// LS Electric XG5000 project: Tip-off System_230829-1
// 기종:PLC_K80S 제목: 회사: 저자: 설명: 
// PLC LSPLC
// module base 0 slot 0: 입출력 모듈:XBM-DN/DP32H2 (DC 24V입력/TR 출력, 32점)
// module base 0 slot 1: 내장위치결정:XBF-PO02E (오픈컬렉터형, 2축)
// module base 0 slot 2: 입력 모듈:XBE-DC16A/B (DC24V 입력, 16점 / DC12/24V 입력, 16점)
// module base 0 slot 3: 입력 모듈:XBE-DC16A/B (DC24V 입력, 16점 / DC12/24V 입력, 16점)
// module base 0 slot 4: 출력 모듈:XBE-RY16A (릴레이 출력, 16점 (2A용, 8점/COM))
// module base 0 slot 5: 출력 모듈:XBE-RY16A (릴레이 출력, 16점 (2A용, 8점/COM))

PROGRAM NewProgram (task: 스캔 프로그램)

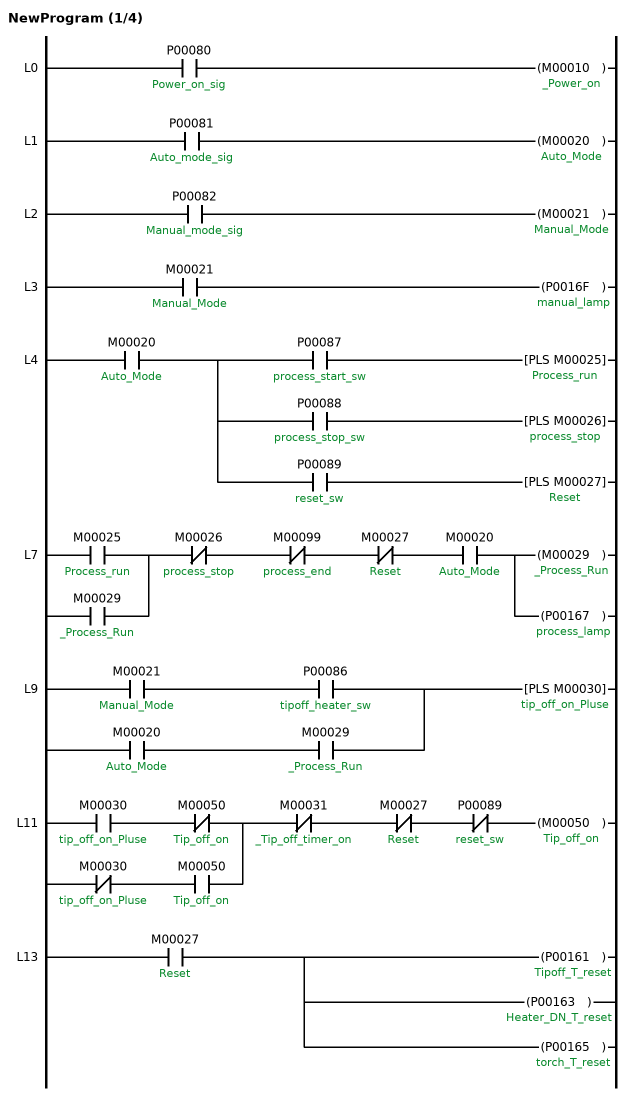
; L0
LOAD      P00080	// Power_on_sig
OUT       M00010	// _Power_on
; L1
LOAD      P00081	// Auto_mode_sig
OUT       M00020	// Auto_Mode
; L2
LOAD      P00082	// Manual_mode_sig
OUT       M00021	// Manual_Mode
; L3
LOAD      M00021	// Manual_Mode
OUT       P0016F	// manual_lamp
; L4
LOAD      M00020	// Auto_Mode
MPUSH
AND       P00087	// process_start_sw
OUTP      M00025	// Process_run
MLOAD
AND       P00088	// process_stop_sw
OUTP      M00026	// process_stop
MPOP
AND       P00089	// reset_sw
OUTP      M00027	// Reset
; L7
LOAD      M00025	// Process_run
OR        M00029	// _Process_Run
AND NOT   M00026	// process_stop
AND NOT   M00099	// process_end
AND NOT   M00027	// Reset
AND       M00020	// Auto_Mode
OUT       M00029	// _Process_Run
OUT       P00167	// process_lamp
; L9
LOAD      M00021	// Manual_Mode
AND       P00086	// tipoff_heater_sw
LOAD      M00020	// Auto_Mode
AND       M00029	// _Process_Run
OR LOAD
OUTP      M00030	// tip_off_on_Pluse
; L11
LOAD      M00030	// tip_off_on_Pluse
AND NOT   M00050	// Tip_off_on
LOAD NOT  M00030	// tip_off_on_Pluse
AND       M00050	// Tip_off_on
OR LOAD
AND NOT   M00031	// _Tip_off_timer_on
AND NOT   M00027	// Reset
AND NOT   P00089	// reset_sw
OUT       M00050	// Tip_off_on
; L13
LOAD      M00027	// Reset
OUT       P00161	// Tipoff_T_reset
OUT       P00163	// Heater_DN_T_reset
OUT       P00165	// torch_T_reset

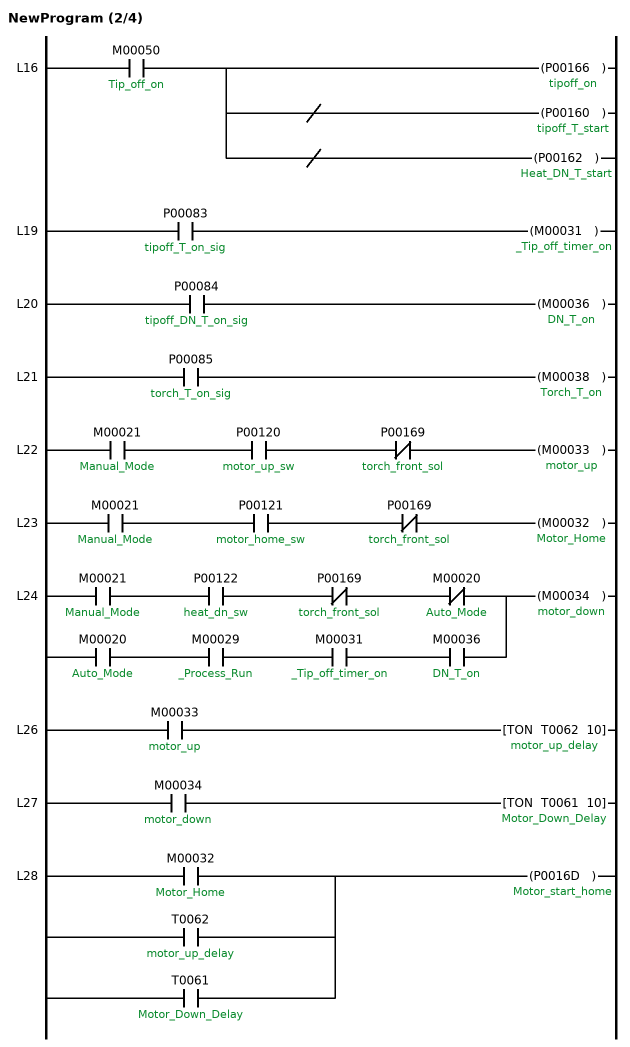
; L16
LOAD      M00050	// Tip_off_on
OUT       P00166	// tipoff_on
MPUSH
NOT
OUT       P00160	// tipoff_T_start
MPOP
NOT
OUT       P00162	// Heat_DN_T_start
; L19
LOAD      P00083	// tipoff_T_on_sig
OUT       M00031	// _Tip_off_timer_on
; L20
LOAD      P00084	// tipoff_DN_T_on_sig
OUT       M00036	// DN_T_on
; L21
LOAD      P00085	// torch_T_on_sig
OUT       M00038	// Torch_T_on
; L22
LOAD      M00021	// Manual_Mode
AND       P00120	// motor_up_sw
AND NOT   P00169	// torch_front_sol
OUT       M00033	// motor_up
; L23
LOAD      M00021	// Manual_Mode
AND       P00121	// motor_home_sw
AND NOT   P00169	// torch_front_sol
OUT       M00032	// Motor_Home
; L24
LOAD      M00021	// Manual_Mode
AND       P00122	// heat_dn_sw
AND NOT   P00169	// torch_front_sol
AND NOT   M00020	// Auto_Mode
LOAD      M00020	// Auto_Mode
AND       M00029	// _Process_Run
AND       M00031	// _Tip_off_timer_on
AND       M00036	// DN_T_on
OR LOAD
OUT       M00034	// motor_down
; L26
LOAD      M00033	// motor_up
TON       T0062 10	// motor_up_delay
; L27
LOAD      M00034	// motor_down
TON       T0061 10	// Motor_Down_Delay
; L28
LOAD      M00032	// Motor_Home
OR        T0062	// motor_up_delay
OR        T0061	// Motor_Down_Delay
OUT       P0016D	// Motor_start_home

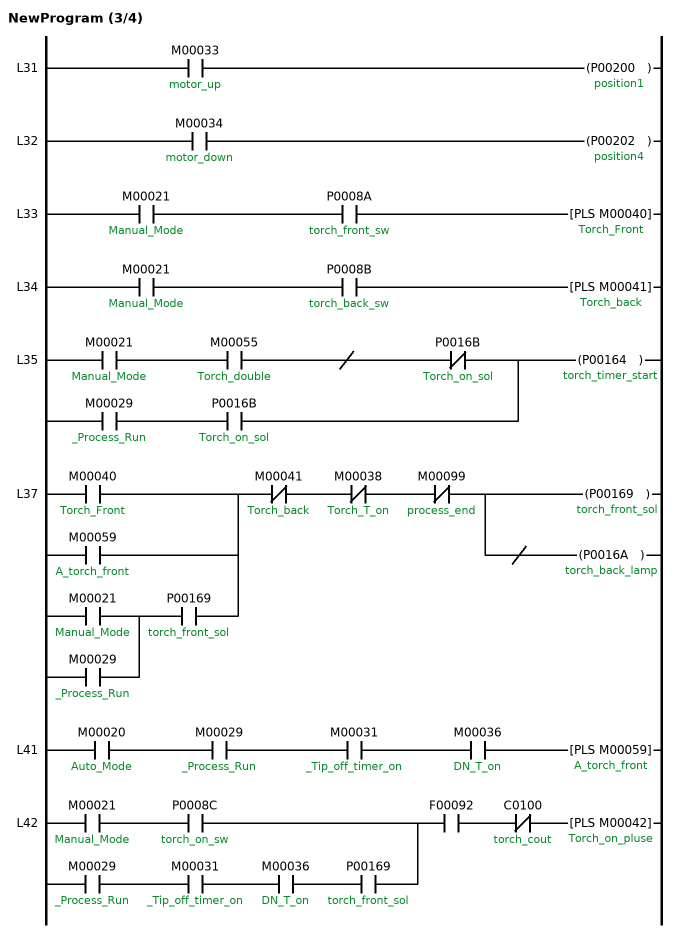
; L31
LOAD      M00033	// motor_up
OUT       P00200	// position1
; L32
LOAD      M00034	// motor_down
OUT       P00202	// position4
; L33
LOAD      M00021	// Manual_Mode
AND       P0008A	// torch_front_sw
OUTP      M00040	// Torch_Front
; L34
LOAD      M00021	// Manual_Mode
AND       P0008B	// torch_back_sw
OUTP      M00041	// Torch_back
; L35
LOAD      M00021	// Manual_Mode
AND       M00055	// Torch_double
NOT
AND NOT   P0016B	// Torch_on_sol
LOAD      M00029	// _Process_Run
AND       P0016B	// Torch_on_sol
OR LOAD
OUT       P00164	// torch_timer_start
; L37
LOAD      M00040	// Torch_Front
OR        M00059	// A_torch_front
LOAD      M00021	// Manual_Mode
OR        M00029	// _Process_Run
AND       P00169	// torch_front_sol
OR LOAD
AND NOT   M00041	// Torch_back
AND NOT   M00038	// Torch_T_on
AND NOT   M00099	// process_end
OUT       P00169	// torch_front_sol
NOT
OUT       P0016A	// torch_back_lamp
; L41
LOAD      M00020	// Auto_Mode
AND       M00029	// _Process_Run
AND       M00031	// _Tip_off_timer_on
AND       M00036	// DN_T_on
OUTP      M00059	// A_torch_front
; L42
LOAD      M00021	// Manual_Mode
AND       P0008C	// torch_on_sw
LOAD      M00029	// _Process_Run
AND       M00031	// _Tip_off_timer_on
AND       M00036	// DN_T_on
AND       P00169	// torch_front_sol
OR LOAD
AND       F00092
AND NOT   C0100	// torch_cout
OUTP      M00042	// Torch_on_pluse

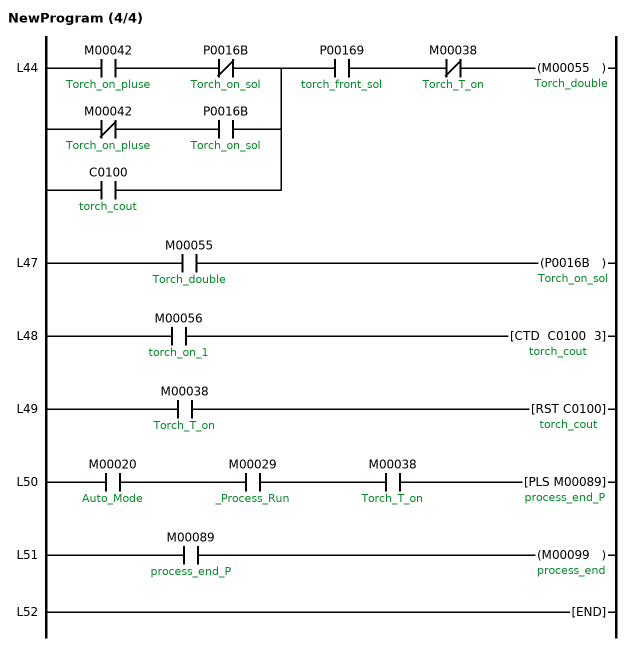
; L44
LOAD      M00042	// Torch_on_pluse
AND NOT   P0016B	// Torch_on_sol
LOAD NOT  M00042	// Torch_on_pluse
AND       P0016B	// Torch_on_sol
OR LOAD
OR        C0100	// torch_cout
AND       P00169	// torch_front_sol
AND NOT   M00038	// Torch_T_on
OUT       M00055	// Torch_double
; L47
LOAD      M00055	// Torch_double
OUT       P0016B	// Torch_on_sol
; L48
LOAD      M00056	// torch_on_1
CTD       C0100 3	// torch_cout
; L49
LOAD      M00038	// Torch_T_on
RST       C0100	// torch_cout
; L50
LOAD      M00020	// Auto_Mode
AND       M00029	// _Process_Run
AND       M00038	// Torch_T_on
OUTP      M00089	// process_end_P
; L51
LOAD      M00089	// process_end_P
OUT       M00099	// process_end
; L52
END

VARIABLES AND COMMENTS (devices not used above)
M00101	BIT	H_L_end
P00100	BIT	H_L_완료
M00105	BIT	H_R_end
T0101	BIT/WORD	H_R_start
M00103	BIT	L_H_end
T0100	BIT/WORD	L_H_start
M00067	BIT	Motor_DN_END
T0060	BIT/WORD	motor_homing_delay
P00055	BIT	motor_out_3
M00063	BIT	Motor_Run_DN_
M00064	BIT	Motor_run_up_
S00201	BIT	motor_step1_up_
S00202	BIT	motor_step2_dn_
S00203	BIT	motor_step3_up_
S00204	BIT	motor_step4_dn_
M00076	BIT	Motor_Strat
P00201	BIT	position2
M00028	BIT	Process_hold
T0081	BIT/WORD	step1_end
T0080	BIT/WORD	step1_start
T0083	BIT/WORD	step2_end
T0082	BIT/WORD	step2_start
T0085	BIT/WORD	step3_end
T0084	BIT/WORD	step3_start
T0087	BIT/WORD	step4_end
T0086	BIT/WORD	step4_start
M00080	BIT	step_start
T0070	BIT/WORD	tilie_H_L_end
M00071	BIT	tilite_Home
M00100	BIT	Tilite_H_L
M00070	BIT	tilite_L
M00102	BIT	Tilite_L_H
P0004D	BIT	Tilit_Home_sol
S00105	BIT	tilte_1_cycle
C0010	BIT/WORD	tilte_2_cycle
M00073	BIT	tilte_count
T0075	BIT/WORD	Tilte_end
P0000E	BIT	tilte_home_sw
S00101	BIT	Tilte_H_L
M00104	BIT	Tilte_H_R
T0072	BIT/WORD	tilte_H_R_end
P0000D	BIT	tilte_Left_sw
S00102	BIT	Tilte_L_H
T0071	BIT/WORD	Tilte_L_H_end
P0004C	BIT	Tilte_L_sol
S00100	BIT	Tilte_reset
M00072	BIT	tilte_right
P0004E	BIT	tilte_right_sol
P0000F	BIT	tilte_right_sw
S00104	BIT	Tilte_R_H
T0073	BIT/WORD	Tilte_R_H_end
M00085	BIT	torch_start
M00035	BIT	Up_Dn_Timer_on
M00062	BIT	_Motor_down
M00060	BIT	_motor_homing
M00061	BIT	_Motor_up
T0090	BIT/WORD	_torch_front
M00090	BIT	_Torch_start
M00066	BIT	__Motor_Down